(* IEC 61131-3 sources: AXOpen/src/integrations/ctrl/src/IntegrationTests/probers, 1 file *)

(* ---- ProbersTest.st ---- *)
USING AXOpen.Core;
USING ix.framework.probers;

NAMESPACE IntegrationTests

CLASS ProbersTestContext EXTENDS AxoContext
    VAR PUBLIC
        ProbeWithCounterTests : ProbeWithCounterTests;
        ProbeWithEndConditionTests : ProberWithCompletedConditionTests;
    END_VAR
    METHOD PROTECTED OVERRIDE Main
        ProbeWithCounterTests.Run(THIS);
        ProbeWithEndConditionTests.Run(THIS);
    END_METHOD
END_CLASS

CLASS ProbeWithCounterTests EXTENDS ProberWithCounterBase
    VAR PUBLIC
        _didExecuteTestMethod : BOOL;
        _numberOfCalls : ULINT;
    END_VAR

    METHOD PROTECTED OVERRIDE Test
        _didExecuteTestMethod := TRUE;
        _numberOfCalls := _numberOfCalls + ULINT#1;
    END_METHOD
END_CLASS

CLASS ProberWithCompletedConditionTests EXTENDS ProberWithCompletedCondition
    VAR PUBLIC
        _didExecuteTestMethod : BOOL;
        _numberOfCalls : ULINT;
    END_VAR

    METHOD PROTECTED OVERRIDE Test  : BOOL
        _didExecuteTestMethod := TRUE;
        _numberOfCalls := ULINT#123;
        Test := TRUE;
    END_METHOD
END_CLASS

END_NAMESPACE
